// SIMATIC S7-200 project (STEP 7-Micro/WIN), CPU 224XP REL 02.01

ORGANIZATION_BLOCK PRINCIPAL:OB1
TITLE=COMENTARIOS DEL PROGRAMA
BEGIN
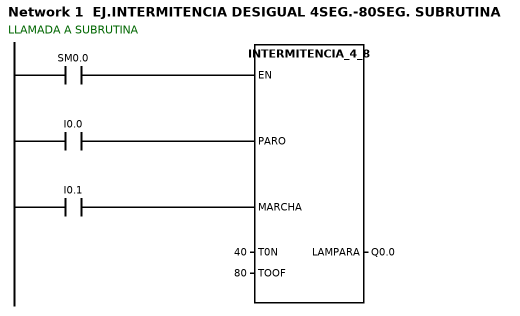
Network 1 // EJ.INTERMITENCIA DESIGUAL 4SEG.-80SEG. SUBRUTINA
// LLAMADA A SUBRUTINA
LD     SM0.0
=      L60.0
LD     I0.0
=      L63.7
LD     I0.1
=      L63.6
LD     L60.0
CALL   INTERMITENCIA_4_8:SBR0, L63.7, L63.6, 40, 80, Q0.0
END_ORGANIZATION_BLOCK

SUBROUTINE_BLOCK INTERMITENCIA_4_8:SBR0
TITLE=COMENTARIOS DE LA SUBRUTINA
VAR_INPUT
PARO:BOOL;	// L0.0 
MARCHA:BOOL;	// L0.1 
T0N:INT;	// LW1 
TOOF:INT;	// LW3 
END_VAR
VAR_OUTPUT
LAMPARA:BOOL;	// L5.0 
END_VAR
VAR
AUXILIAR_2:BOOL;	// L5.1 
END_VAR
BEGIN
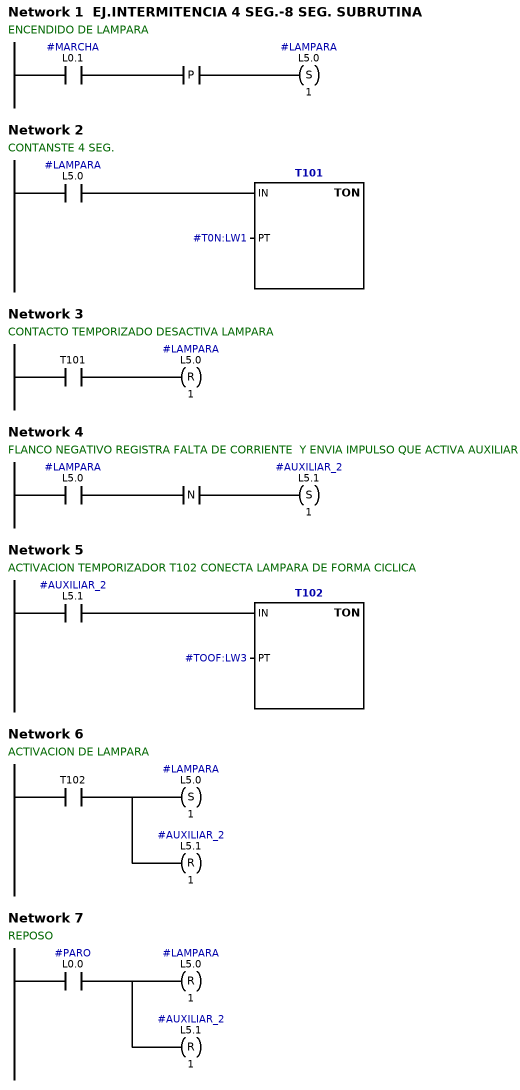
Network 1 // EJ.INTERMITENCIA 4 SEG.-8 SEG. SUBRUTINA
// ENCENDIDO DE LAMPARA
LD     #MARCHA:L0.1
EU
S      #LAMPARA:L5.0, 1
Network 2
// CONTANSTE 4 SEG.
LD     #LAMPARA:L5.0
TON    T101, #T0N:LW1
Network 3
// CONTACTO TEMPORIZADO DESACTIVA LAMPARA
LD     T101
R      #LAMPARA:L5.0, 1
Network 4
// FLANCO NEGATIVO REGISTRA FALTA DE CORRIENTE  Y ENVIA IMPULSO QUE ACTIVA AUXILIAR 2
LD     #LAMPARA:L5.0
ED
S      #AUXILIAR_2:L5.1, 1
Network 5
// ACTIVACION TEMPORIZADOR T102 CONECTA LAMPARA DE FORMA CICLICA
LD     #AUXILIAR_2:L5.1
TON    T102, #TOOF:LW3
Network 6
// ACTIVACION DE LAMPARA 
LD     T102
S      #LAMPARA:L5.0, 1
R      #AUXILIAR_2:L5.1, 1
Network 7
// REPOSO
LD     #PARO:L0.0
R      #LAMPARA:L5.0, 1
R      #AUXILIAR_2:L5.1, 1
END_SUBROUTINE_BLOCK
